Fanuc KAREL source: PEND_SEMA.kl

PROGRAM T
%NOLOCKGROUP
VAR
 v0 : INTEGER
 v1 : INTEGER
 v2 : BOOLEAN
BEGIN
 PEND_SEMA(v0, v1, v2)
END T
